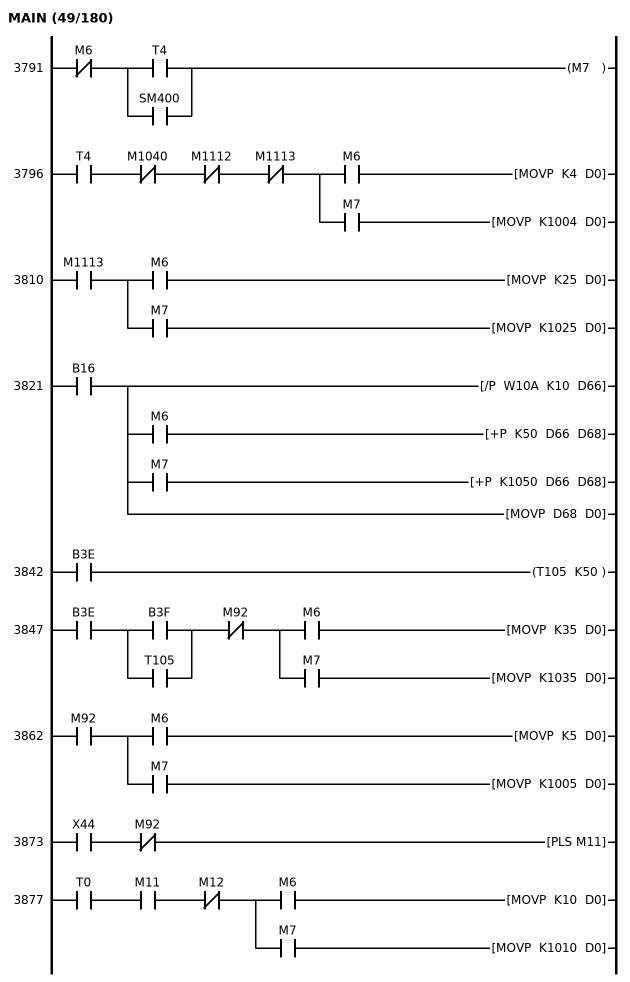
[picture p48: ladder of MAIN, rungs at steps 3791 to 3877]
3791  LDI     M6
      LD      T4
      OR      SM400
      ANB
      OUT     M7
3796  LD      T4
      ANI     M1040
      ANI     M1112
      ANI     M1113
      MPS
      AND     M6
      MOVP    K4 D0
      MPP
      AND     M7
      MOVP    K1004 D0
3810  LD      M1113
      MPS
      AND     M6
      MOVP    K25 D0
      MPP
      AND     M7
      MOVP    K1025 D0
3821  LD      B16
      /P      W10A K10 D66
      MPS
      AND     M6
      +P      K50 D66 D68
      MRD
      AND     M7
      +P      K1050 D66 D68
      MPP
      MOVP    D68 D0
3842  LD      B3E
      OUT     T105 K50
3847  LD      B3E
      LD      B3F
      OR      T105
      ANB
      ANI     M92
      MPS
      AND     M6
      MOVP    K35 D0
      MPP
      AND     M7
      MOVP    K1035 D0
3862  LD      M92
      MPS
      AND     M6
      MOVP    K5 D0
      MPP
      AND     M7
      MOVP    K1005 D0
3873  LD      X44
      ANI     M92
      PLS     M11
3877  LD      T0
      AND     M11
      ANI     M12
      MPS
      AND     M6
      MOVP    K10 D0
      MPP
      AND     M7
      MOVP    K1010 D0
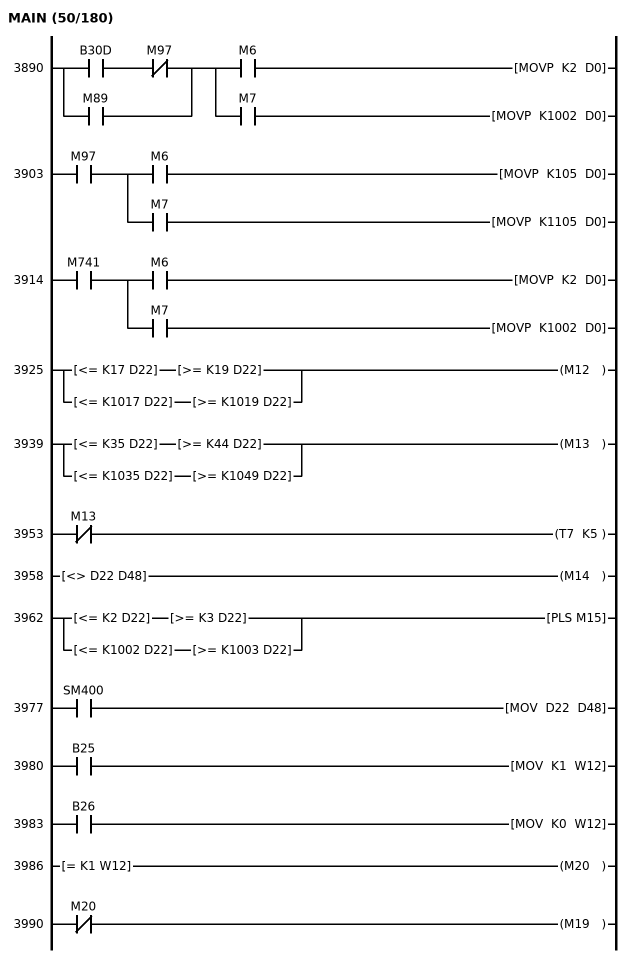
3890  LD      B30D
      ANI     M97
      OR      M89
      MPS
      AND     M6
      MOVP    K2 D0
      MPP
      AND     M7
      MOVP    K1002 D0
3903  LD      M97
      MPS
      AND     M6
      MOVP    K105 D0
      MPP
      AND     M7
      MOVP    K1105 D0
3914  LD      M741
      MPS
      AND     M6
      MOVP    K2 D0
      MPP
      AND     M7
      MOVP    K1002 D0
3925  LD<=    K17 D22
      AND>=   K19 D22
      LD<=    K1017 D22
      AND>=   K1019 D22
      ORB
      OUT     M12
3939  LD<=    K35 D22
      AND>=   K44 D22
      LD<=    K1035 D22
      AND>=   K1049 D22
      ORB
      OUT     M13
3953  LDI     M13
      OUT     T7 K5
3958  LD<>    D22 D48
      OUT     M14
3962  LD<=    K2 D22
      AND>=   K3 D22
      LD<=    K1002 D22
      AND>=   K1003 D22
      ORB
      PLS     M15
3977  LD      SM400
      MOV     D22 D48
3980  LD      B25
      MOV     K1 W12
3983  LD      B26
      MOV     K0 W12
3986  LD=     K1 W12
      OUT     M20
3990  LDI     M20
      OUT     M19
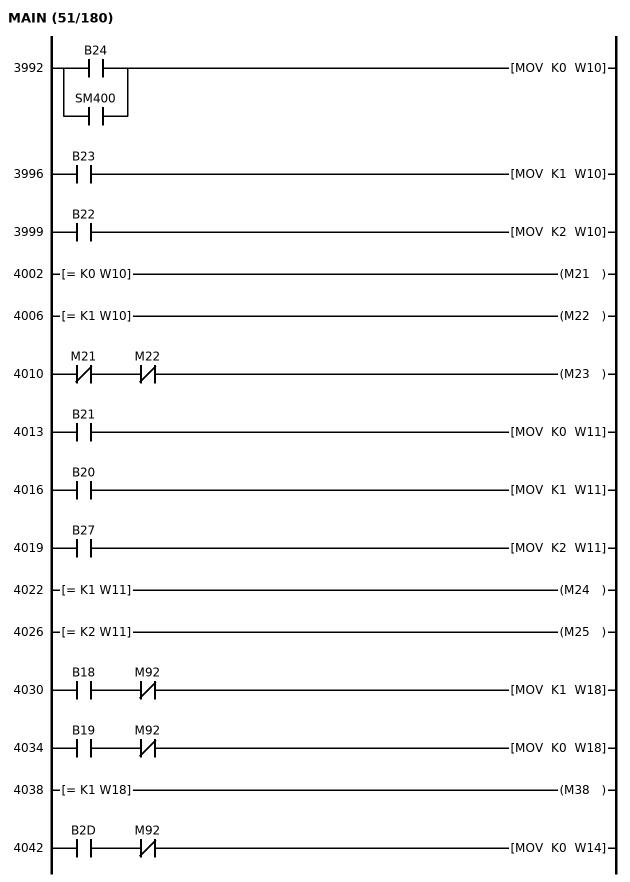
3992  LD      B24
      OR      SM400
      MOV     K0 W10
3996  LD      B23
      MOV     K1 W10
3999  LD      B22
      MOV     K2 W10
4002  LD=     K0 W10
      OUT     M21
4006  LD=     K1 W10
      OUT     M22
4010  LDI     M21
      ANI     M22
      OUT     M23
4013  LD      B21
      MOV     K0 W11
4016  LD      B20
      MOV     K1 W11
4019  LD      B27
      MOV     K2 W11
4022  LD=     K1 W11
      OUT     M24
4026  LD=     K2 W11
      OUT     M25
4030  LD      B18
      ANI     M92
      MOV     K1 W18
4034  LD      B19
      ANI     M92
      MOV     K0 W18
4038  LD=     K1 W18
      OUT     M38
4042  LD      B2D
      ANI     M92
      MOV     K0 W14
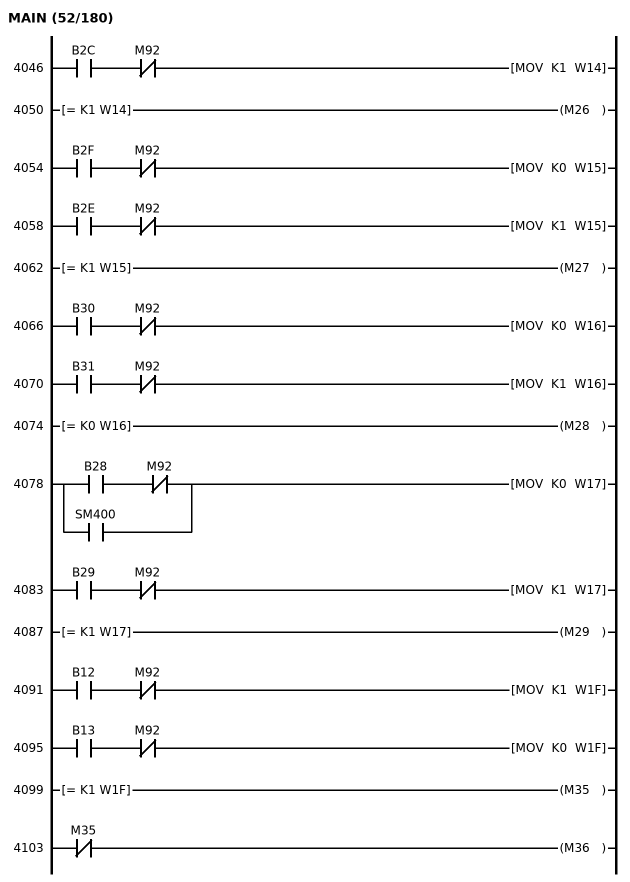
4046  LD      B2C
      ANI     M92
      MOV     K1 W14
4050  LD=     K1 W14
      OUT     M26
4054  LD      B2F
      ANI     M92
      MOV     K0 W15
4058  LD      B2E
      ANI     M92
      MOV     K1 W15
4062  LD=     K1 W15
      OUT     M27
4066  LD      B30
      ANI     M92
      MOV     K0 W16
4070  LD      B31
      ANI     M92
      MOV     K1 W16
4074  LD=     K0 W16
      OUT     M28
4078  LD      B28
      ANI     M92
      OR      SM400
      MOV     K0 W17
4083  LD      B29
      ANI     M92
      MOV     K1 W17
4087  LD=     K1 W17
      OUT     M29
4091  LD      B12
      ANI     M92
      MOV     K1 W1F
4095  LD      B13
      ANI     M92
      MOV     K0 W1F
4099  LD=     K1 W1F
      OUT     M35
4103  LDI     M35
      OUT     M36
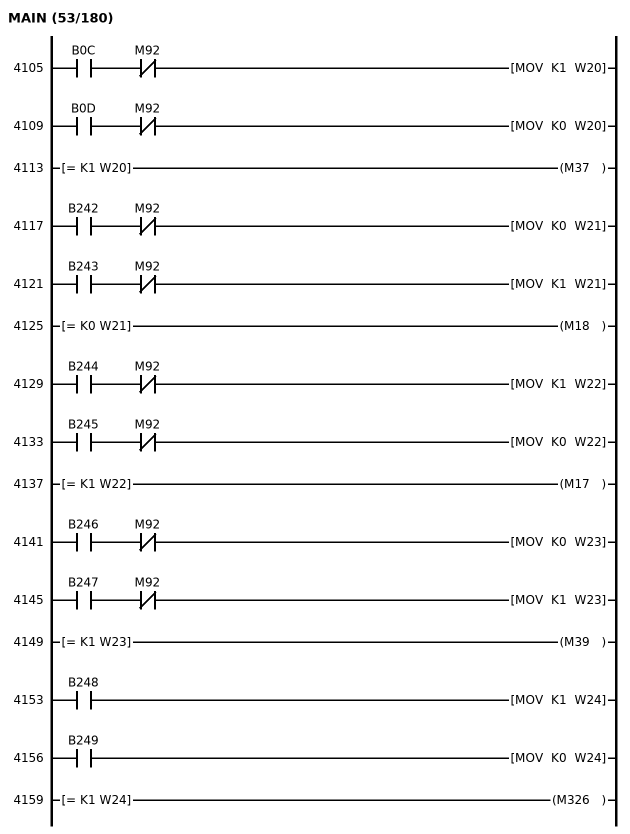
4105  LD      B0C
      ANI     M92
      MOV     K1 W20
4109  LD      B0D
      ANI     M92
      MOV     K0 W20
4113  LD=     K1 W20
      OUT     M37
4117  LD      B242
      ANI     M92
      MOV     K0 W21
4121  LD      B243
      ANI     M92
      MOV     K1 W21
4125  LD=     K0 W21
      OUT     M18
4129  LD      B244
      ANI     M92
      MOV     K1 W22
4133  LD      B245
      ANI     M92
      MOV     K0 W22
4137  LD=     K1 W22
      OUT     M17
4141  LD      B246
      ANI     M92
      MOV     K0 W23
4145  LD      B247
      ANI     M92
      MOV     K1 W23
4149  LD=     K1 W23
      OUT     M39
4153  LD      B248
      MOV     K1 W24
4156  LD      B249
      MOV     K0 W24
4159  LD=     K1 W24
      OUT     M326
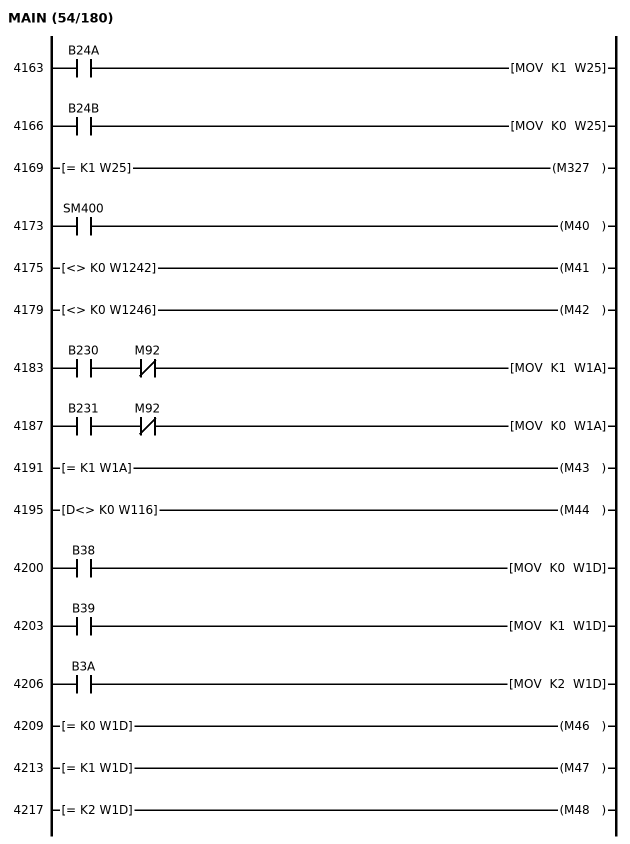
4163  LD      B24A
      MOV     K1 W25
4166  LD      B24B
      MOV     K0 W25
4169  LD=     K1 W25
      OUT     M327
4173  LD      SM400
      OUT     M40
4175  LD<>    K0 W1242
      OUT     M41
4179  LD<>    K0 W1246
      OUT     M42
4183  LD      B230
      ANI     M92
      MOV     K1 W1A
4187  LD      B231
      ANI     M92
      MOV     K0 W1A
4191  LD=     K1 W1A
      OUT     M43
4195  LDD<>   K0 W116
      OUT     M44
4200  LD      B38
      MOV     K0 W1D
4203  LD      B39
      MOV     K1 W1D
4206  LD      B3A
      MOV     K2 W1D
4209  LD=     K0 W1D
      OUT     M46
4213  LD=     K1 W1D
      OUT     M47
4217  LD=     K2 W1D
      OUT     M48
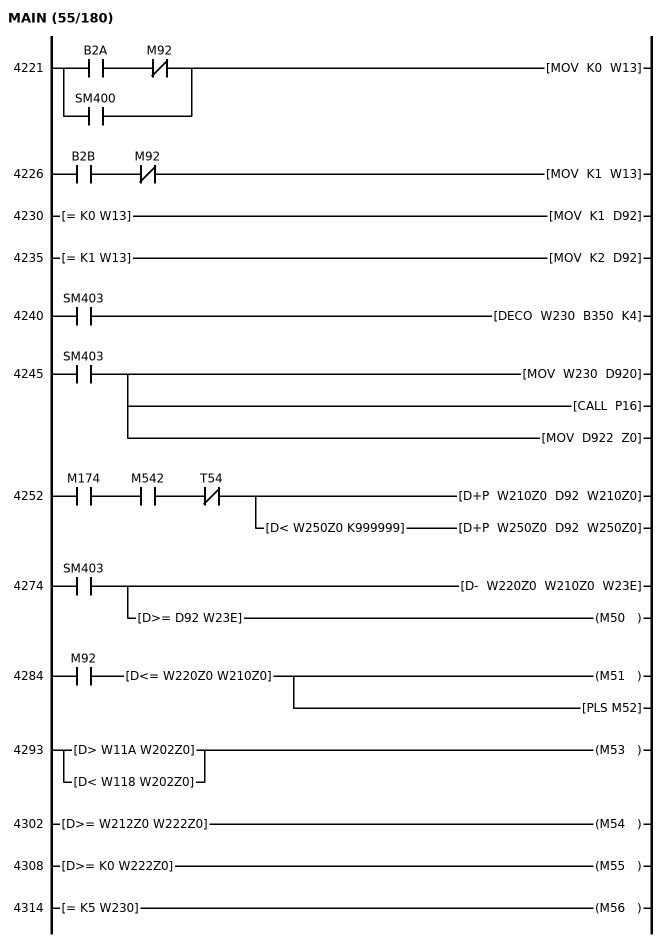
4221  LD      B2A
      ANI     M92
      OR      SM400
      MOV     K0 W13
4226  LD      B2B
      ANI     M92
      MOV     K1 W13
4230  LD=     K0 W13
      MOV     K1 D92
4235  LD=     K1 W13
      MOV     K2 D92
4240  LD      SM403
      DECO    W230 B350 K4
4245  LD      SM403
      MOV     W230 D920
      CALL    P16
      MOV     D922 Z0
4252  LD      M174
      AND     M542
      ANI     T54
      D+P     W210Z0 D92 W210Z0
      ANDD<   W250Z0 K999999
      D+P     W250Z0 D92 W250Z0
4274  LD      SM403
      D-      W220Z0 W210Z0 W23E
      ANDD>=  D92 W23E
      OUT     M50
4284  LD      M92
      ANDD<=  W220Z0 W210Z0
      OUT     M51
      PLS     M52
4293  LDD>    W11A W202Z0
      ORD<    W118 W202Z0
      OUT     M53
4302  LDD>=   W212Z0 W222Z0
      OUT     M54
4308  LDD>=   K0 W222Z0
      OUT     M55
4314  LD=     K5 W230
      OUT     M56
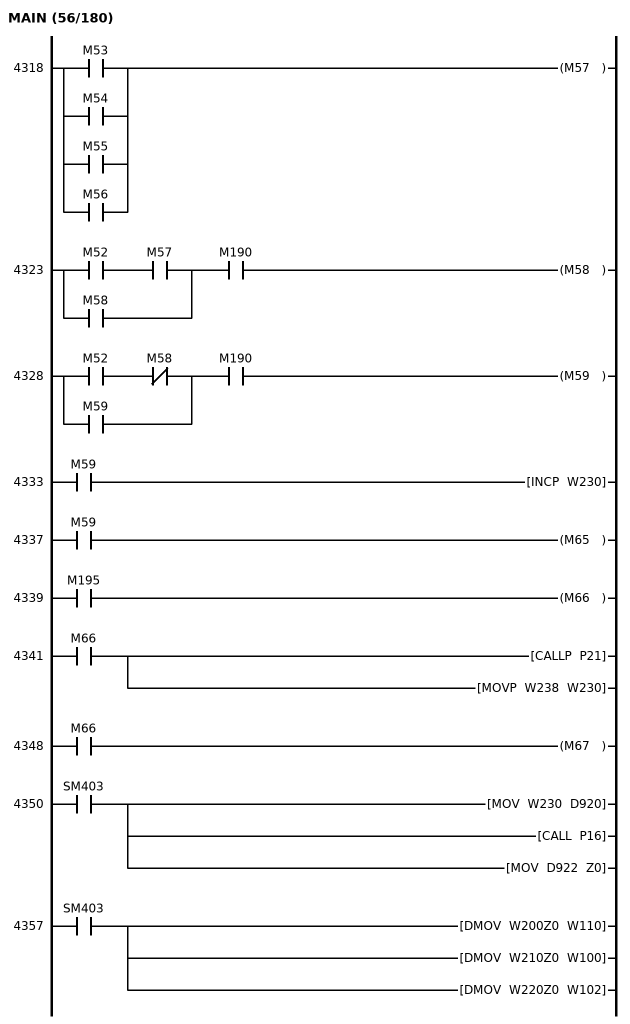
4318  LD      M53
      OR      M54
      OR      M55
      OR      M56
      OUT     M57
4323  LD      M52
      AND     M57
      OR      M58
      AND     M190
      OUT     M58
4328  LD      M52
      ANI     M58
      OR      M59
      AND     M190
      OUT     M59
4333  LD      M59
      INCP    W230
4337  LD      M59
      OUT     M65
4339  LD      M195
      OUT     M66
4341  LD      M66
      CALLP   P21
      MOVP    W238 W230
4348  LD      M66
      OUT     M67
4350  LD      SM403
      MOV     W230 D920
      CALL    P16
      MOV     D922 Z0
4357  LD      SM403
      DMOV    W200Z0 W110
      DMOV    W210Z0 W100
      DMOV    W220Z0 W102
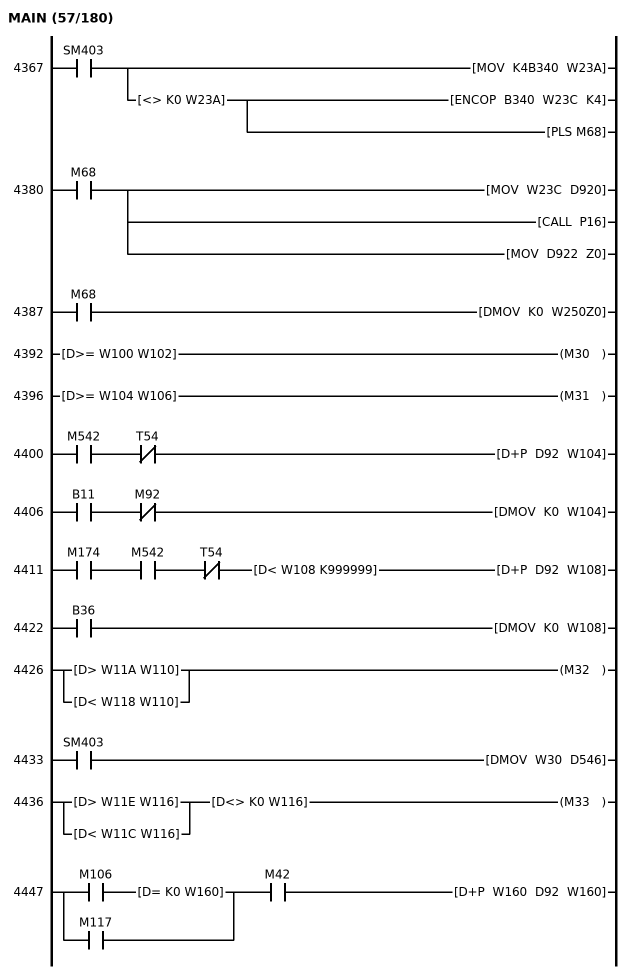
4367  LD      SM403
      MOV     K4B340 W23A
      AND<>   K0 W23A
      ENCOP   B340 W23C K4
      PLS     M68
4380  LD      M68
      MOV     W23C D920
      CALL    P16
      MOV     D922 Z0
4387  LD      M68
      DMOV    K0 W250Z0
4392  LDD>=   W100 W102
      OUT     M30
4396  LDD>=   W104 W106
      OUT     M31
4400  LD      M542
      ANI     T54
      D+P     D92 W104
4406  LD      B11
      ANI     M92
      DMOV    K0 W104
4411  LD      M174
      AND     M542
      ANI     T54
      ANDD<   W108 K999999
      D+P     D92 W108
4422  LD      B36
      DMOV    K0 W108
4426  LDD>    W11A W110
      ORD<    W118 W110
      OUT     M32
4433  LD      SM403
      DMOV    W30 D546
4436  LDD>    W11E W116
      ORD<    W11C W116
      ANDD<>  K0 W116
      OUT     M33
4447  LD      M106
      ANDD=   K0 W160
      OR      M117
      AND     M42
      D+P     W160 D92 W160
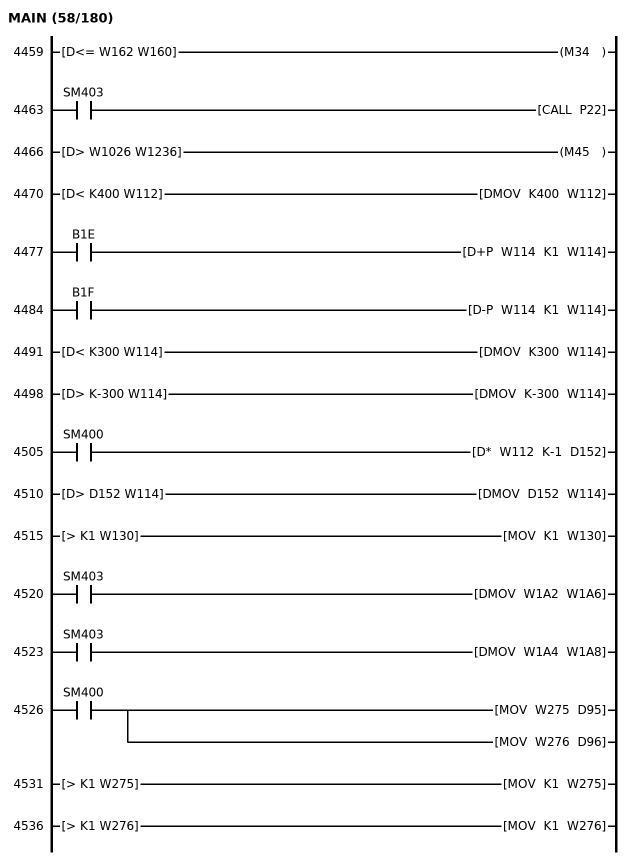
4459  LDD<=   W162 W160
      OUT     M34
4463  LD      SM403
      CALL    P22
4466  LDD>    W1026 W1236
      OUT     M45
4470  LDD<    K400 W112
      DMOV    K400 W112
4477  LD      B1E
      D+P     W114 K1 W114
4484  LD      B1F
      D-P     W114 K1 W114
4491  LDD<    K300 W114
      DMOV    K300 W114
4498  LDD>    K-300 W114
      DMOV    K-300 W114
4505  LD      SM400
      D*      W112 K-1 D152
4510  LDD>    D152 W114
      DMOV    D152 W114
4515  LD>     K1 W130
      MOV     K1 W130
4520  LD      SM403
      DMOV    W1A2 W1A6
4523  LD      SM403
      DMOV    W1A4 W1A8
4526  LD      SM400
      MOV     W275 D95
      MOV     W276 D96
4531  LD>     K1 W275
      MOV     K1 W275
4536  LD>     K1 W276
      MOV     K1 W276
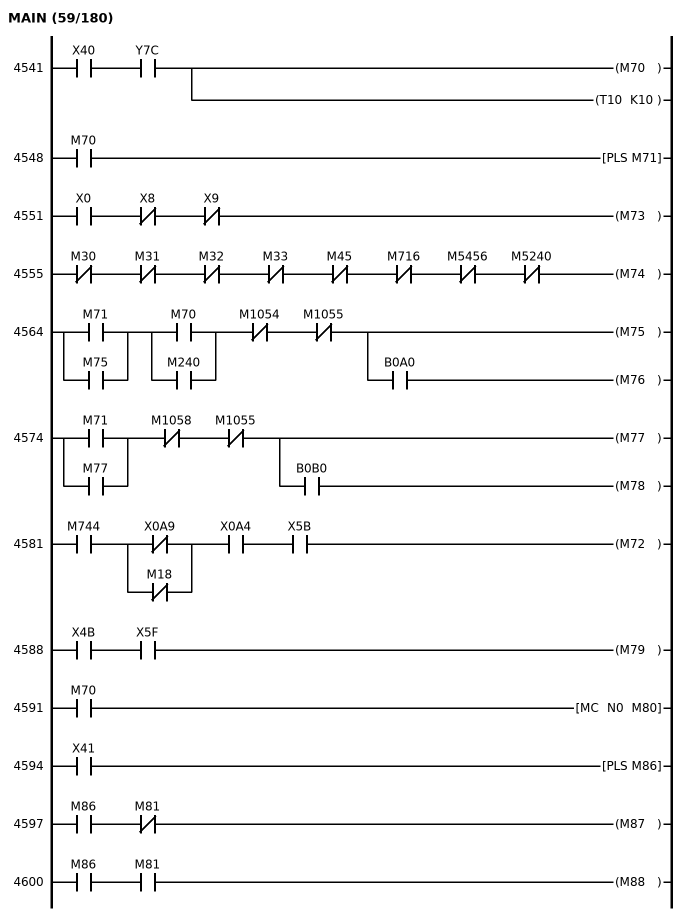
4541  LD      X40
      AND     Y7C
      OUT     M70
      OUT     T10 K10
4548  LD      M70
      PLS     M71
4551  LD      X0
      ANI     X8
      ANI     X9
      OUT     M73
4555  LDI     M30
      ANI     M31
      ANI     M32
      ANI     M33
      ANI     M45
      ANI     M716
      ANI     M5456
      ANI     M5240
      OUT     M74
4564  LD      M71
      OR      M75
      LD      M70
      OR      M240
      ANB
      ANI     M1054
      ANI     M1055
      OUT     M75
      AND     B0A0
      OUT     M76
4574  LD      M71
      OR      M77
      ANI     M1058
      ANI     M1055
      OUT     M77
      AND     B0B0
      OUT     M78
4581  LD      M744
      LDI     X0A9
      ORI     M18
      ANB
      AND     X0A4
      AND     X5B
      OUT     M72
4588  LD      X4B
      AND     X5F
      OUT     M79
4591  LD      M70
      MC      N0 M80
4594  LD      X41
      PLS     M86
4597  LD      M86
      ANI     M81
      OUT     M87
4600  LD      M86
      AND     M81
      OUT     M88
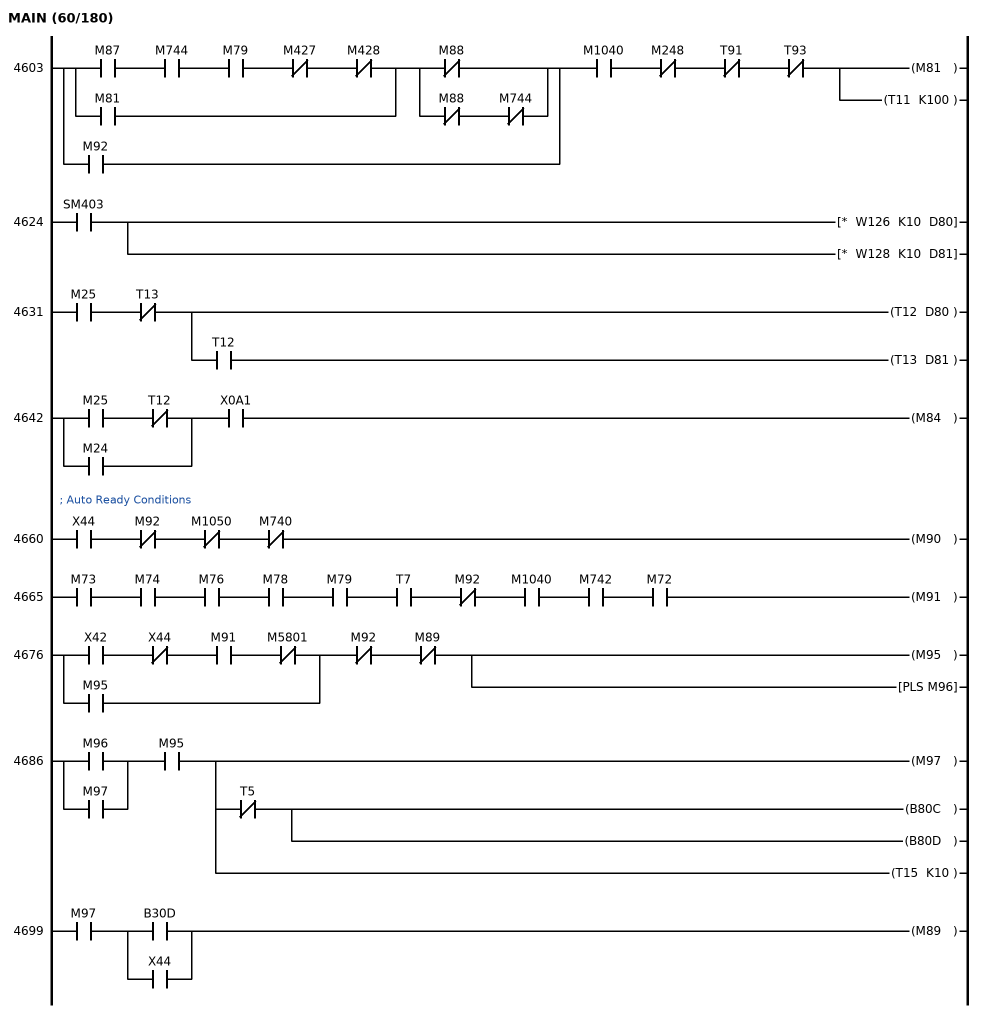
4603  LD      M87
      AND     M744
      AND     M79
      ANI     M427
      ANI     M428
      OR      M81
      LDI     M88
      LDI     M88
      ANI     M744
      ORB
      ANB
      OR      M92
      AND     M1040
      ANI     M248
      ANI     T91
      ANI     T93
      OUT     M81
      OUT     T11 K100
4624  LD      SM403
      *       W126 K10 D80
      *       W128 K10 D81
4631  LD      M25
      ANI     T13
      OUT     T12 D80
      AND     T12
      OUT     T13 D81
4642  LD      M25
      ANI     T12
      OR      M24
      AND     X0A1
      OUT     M84
; Auto Ready Conditions
4660  LD      X44
      ANI     M92
      ANI     M1050
      ANI     M740
      OUT     M90
4665  LD      M73
      AND     M74
      AND     M76
      AND     M78
      AND     M79
      AND     T7
      ANI     M92
      AND     M1040
      AND     M742
      AND     M72
      OUT     M91
4676  LD      X42
      ANI     X44
      AND     M91
      ANI     M5801
      OR      M95
      ANI     M92
      ANI     M89
      OUT     M95
      PLS     M96
4686  LD      M96
      OR      M97
      AND     M95
      OUT     M97
      MPS
      ANI     T5
      OUT     B80C
      OUT     B80D
      MPP
      OUT     T15 K10
4699  LD      M97
      LD      B30D
      OR      X44
      ANB
      OUT     M89
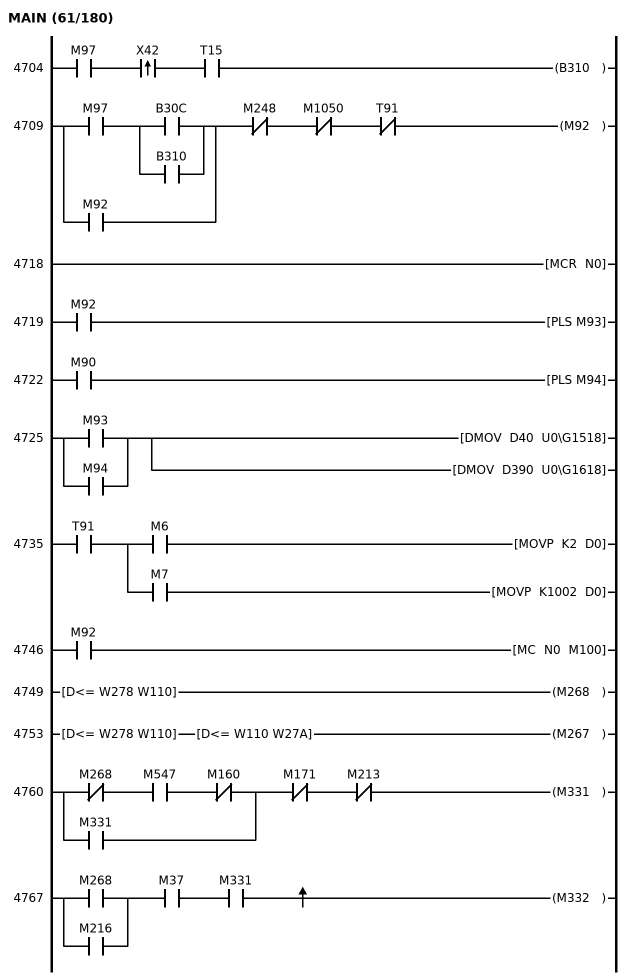
4704  LD      M97
      ANDP    X42
      AND     T15
      OUT     B310
4709  LD      M97
      LD      B30C
      OR      B310
      ANB
      OR      M92
      ANI     M248
      ANI     M1050
      ANI     T91
      OUT     M92
4718  MCR     N0
4719  LD      M92
      PLS     M93
4722  LD      M90
      PLS     M94
4725  LD      M93
      OR      M94
      DMOV    D40 U0\G1518
      DMOV    D390 U0\G1618
4735  LD      T91
      MPS
      AND     M6
      MOVP    K2 D0
      MPP
      AND     M7
      MOVP    K1002 D0
4746  LD      M92
      MC      N0 M100
4749  LDD<=   W278 W110
      OUT     M268
4753  LDD<=   W278 W110
      ANDD<=  W110 W27A
      OUT     M267
4760  LDI     M268
      AND     M547
      ANI     M160
      OR      M331
      ANI     M171
      ANI     M213
      OUT     M331
4767  LD      M268
      OR      M216
      AND     M37
      AND     M331
      MEP
      OUT     M332
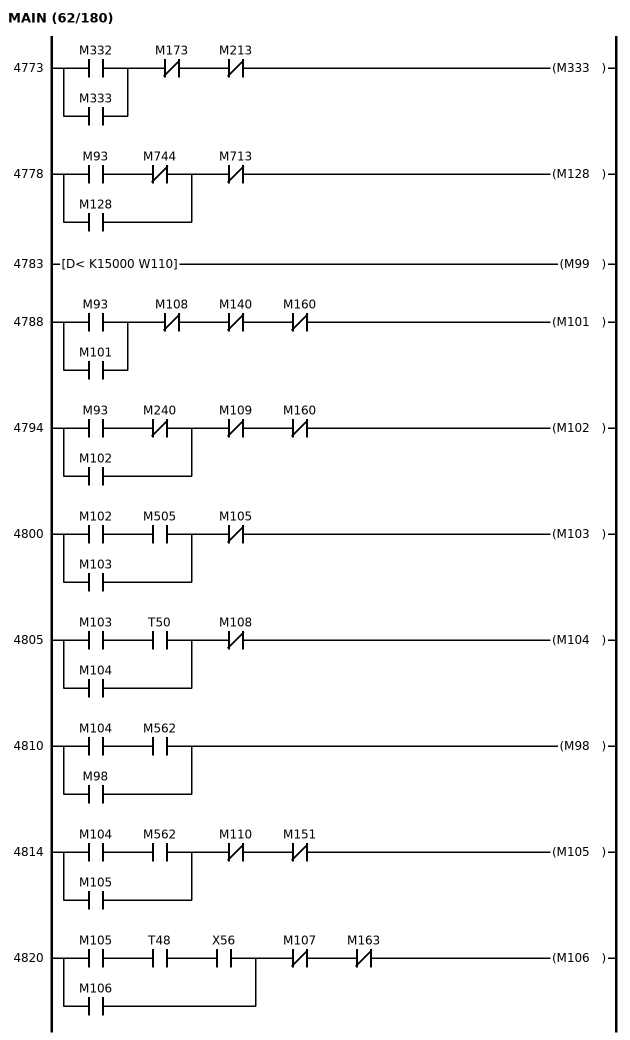
4773  LD      M332
      OR      M333
      ANI     M173
      ANI     M213
      OUT     M333
4778  LD      M93
      ANI     M744
      OR      M128
      ANI     M713
      OUT     M128
4783  LDD<    K15000 W110
      OUT     M99
4788  LD      M93
      OR      M101
      ANI     M108
      ANI     M140
      ANI     M160
      OUT     M101
4794  LD      M93
      ANI     M240
      OR      M102
      ANI     M109
      ANI     M160
      OUT     M102
4800  LD      M102
      AND     M505
      OR      M103
      ANI     M105
      OUT     M103
4805  LD      M103
      AND     T50
      OR      M104
      ANI     M108
      OUT     M104
4810  LD      M104
      AND     M562
      OR      M98
      OUT     M98
4814  LD      M104
      AND     M562
      OR      M105
      ANI     M110
      ANI     M151
      OUT     M105
4820  LD      M105
      AND     T48
      AND     X56
      OR      M106
      ANI     M107
      ANI     M163
      OUT     M106
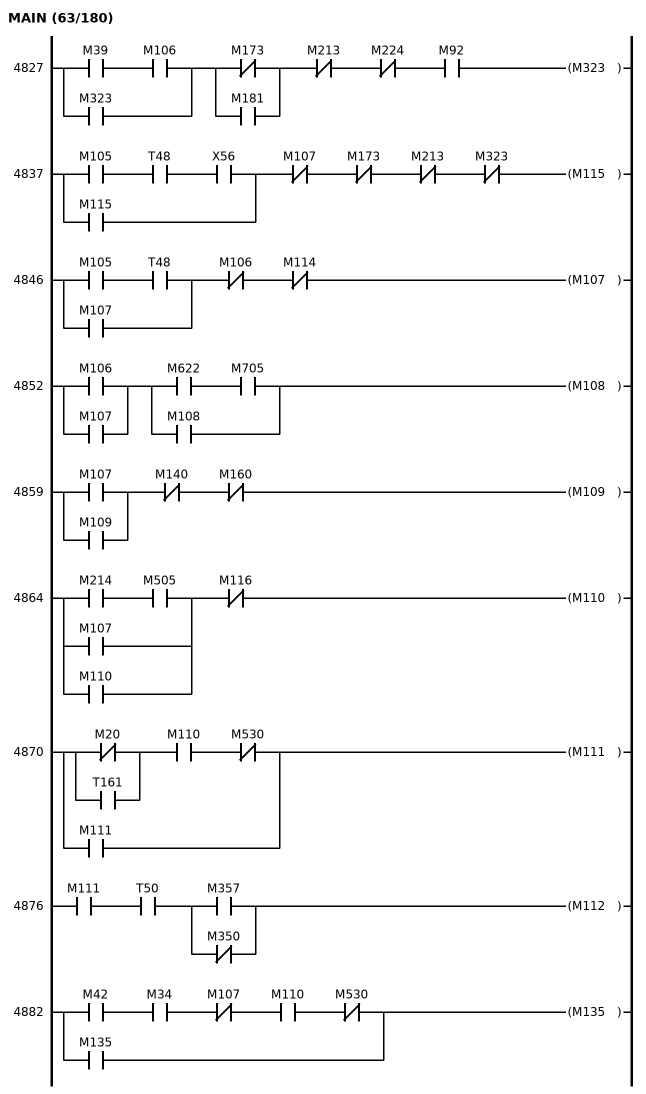
4827  LD      M39
      AND     M106
      OR      M323
      LDI     M173
      OR      M181
      ANB
      ANI     M213
      ANI     M224
      AND     M92
      OUT     M323
4837  LD      M105
      AND     T48
      AND     X56
      OR      M115
      ANI     M107
      ANI     M173
      ANI     M213
      ANI     M323
      OUT     M115
4846  LD      M105
      AND     T48
      OR      M107
      ANI     M106
      ANI     M114
      OUT     M107
4852  LD      M106
      OR      M107
      LD      M622
      AND     M705
      OR      M108
      ANB
      OUT     M108
4859  LD      M107
      OR      M109
      ANI     M140
      ANI     M160
      OUT     M109
4864  LD      M214
      AND     M505
      OR      M107
      OR      M110
      ANI     M116
      OUT     M110
4870  LDI     M20
      OR      T161
      AND     M110
      ANI     M530
      OR      M111
      OUT     M111
4876  LD      M111
      AND     T50
      LD      M357
      ORI     M350
      ANB
      OUT     M112
4882  LD      M42
      AND     M34
      ANI     M107
      AND     M110
      ANI     M530
      OR      M135
      OUT     M135
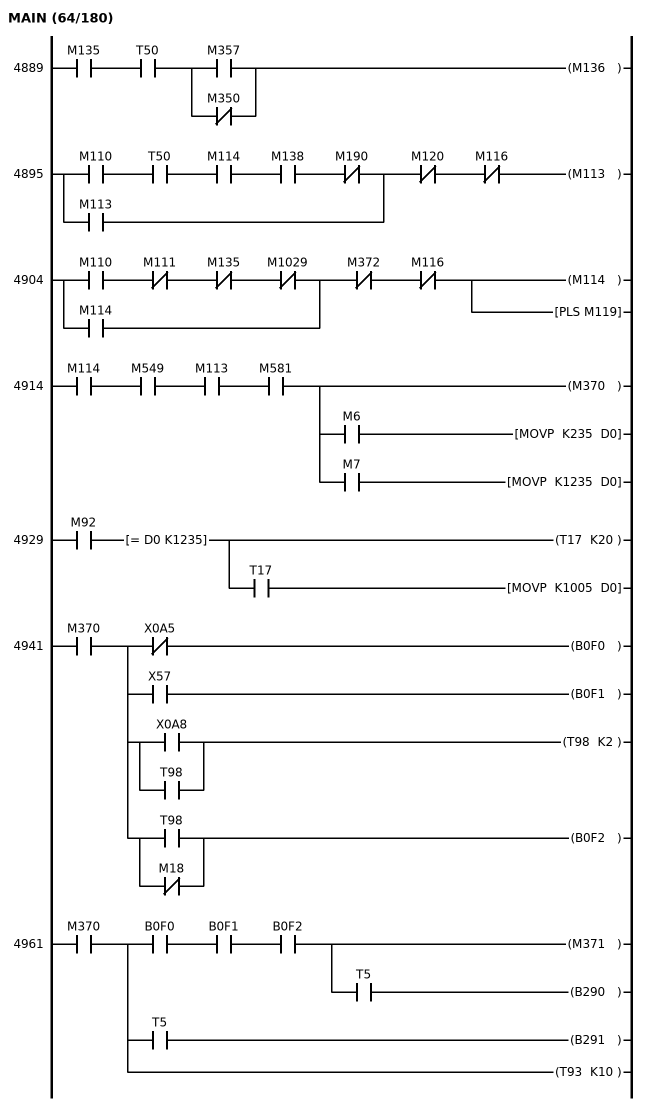
4889  LD      M135
      AND     T50
      LD      M357
      ORI     M350
      ANB
      OUT     M136
4895  LD      M110
      AND     T50
      AND     M114
      AND     M138
      ANI     M190
      OR      M113
      ANI     M120
      ANI     M116
      OUT     M113
4904  LD      M110
      ANI     M111
      ANI     M135
      ANI     M1029
      OR      M114
      ANI     M372
      ANI     M116
      OUT     M114
      PLS     M119
4914  LD      M114
      AND     M549
      AND     M113
      AND     M581
      OUT     M370
      MPS
      AND     M6
      MOVP    K235 D0
      MPP
      AND     M7
      MOVP    K1235 D0
4929  LD      M92
      AND=    D0 K1235
      OUT     T17 K20
      AND     T17
      MOVP    K1005 D0
4941  LD      M370
      MPS
      ANI     X0A5
      OUT     B0F0
      MRD
      AND     X57
      OUT     B0F1
      MRD
      LD      X0A8
      OR      T98
      ANB
      OUT     T98 K2
      MPP
      LD      T98
      ORI     M18
      ANB
      OUT     B0F2
4961  LD      M370
      MPS
      AND     B0F0
      AND     B0F1
      AND     B0F2
      OUT     M371
      AND     T5
      OUT     B290
      MRD
      AND     T5
      OUT     B291
      MPP
      OUT     T93 K10
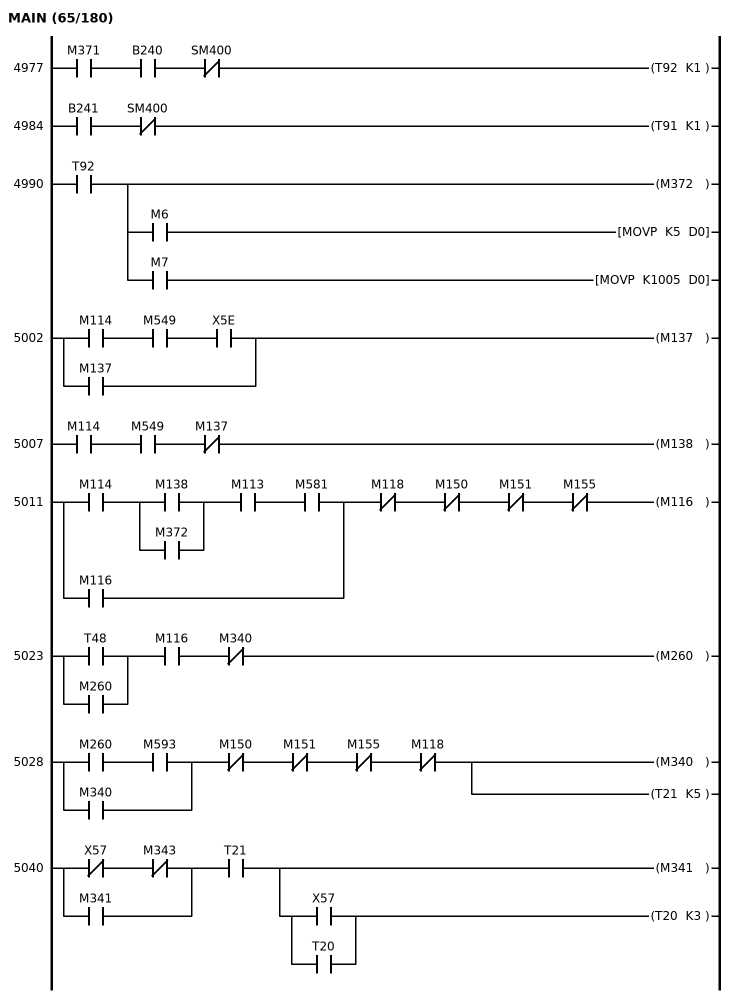
4977  LD      M371
      AND     B240
      ANI     SM400
      OUT     T92 K1
4984  LD      B241
      ANI     SM400
      OUT     T91 K1
4990  LD      T92
      OUT     M372
      MPS
      AND     M6
      MOVP    K5 D0
      MPP
      AND     M7
      MOVP    K1005 D0
5002  LD      M114
      AND     M549
      AND     X5E
      OR      M137
      OUT     M137
5007  LD      M114
      AND     M549
      ANI     M137
      OUT     M138
5011  LD      M114
      LD      M138
      OR      M372
      ANB
      AND     M113
      AND     M581
      OR      M116
      ANI     M118
      ANI     M150
      ANI     M151
      ANI     M155
      OUT     M116
5023  LD      T48
      OR      M260
      AND     M116
      ANI     M340
      OUT     M260
5028  LD      M260
      AND     M593
      OR      M340
      ANI     M150
      ANI     M151
      ANI     M155
      ANI     M118
      OUT     M340
      OUT     T21 K5
5040  LDI     X57
      ANI     M343
      OR      M341
      AND     T21
      OUT     M341
      LD      X57
      OR      T20
      ANB
      OUT     T20 K3
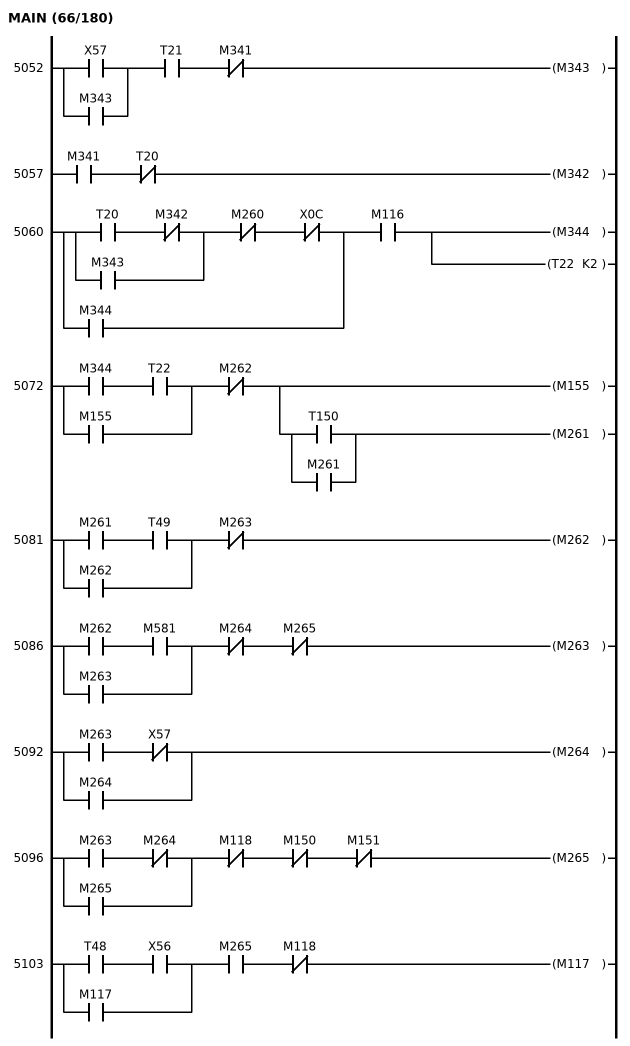
5052  LD      X57
      OR      M343
      AND     T21
      ANI     M341
      OUT     M343
5057  LD      M341
      ANI     T20
      OUT     M342
5060  LD      T20
      ANI     M342
      OR      M343
      ANI     M260
      ANI     X0C
      OR      M344
      AND     M116
      OUT     M344
      OUT     T22 K2
5072  LD      M344
      AND     T22
      OR      M155
      ANI     M262
      OUT     M155
      LD      T150
      OR      M261
      ANB
      OUT     M261
5081  LD      M261
      AND     T49
      OR      M262
      ANI     M263
      OUT     M262
5086  LD      M262
      AND     M581
      OR      M263
      ANI     M264
      ANI     M265
      OUT     M263
5092  LD      M263
      ANI     X57
      OR      M264
      OUT     M264
5096  LD      M263
      ANI     M264
      OR      M265
      ANI     M118
      ANI     M150
      ANI     M151
      OUT     M265
5103  LD      T48
      AND     X56
      OR      M117
      AND     M265
      ANI     M118
      OUT     M117
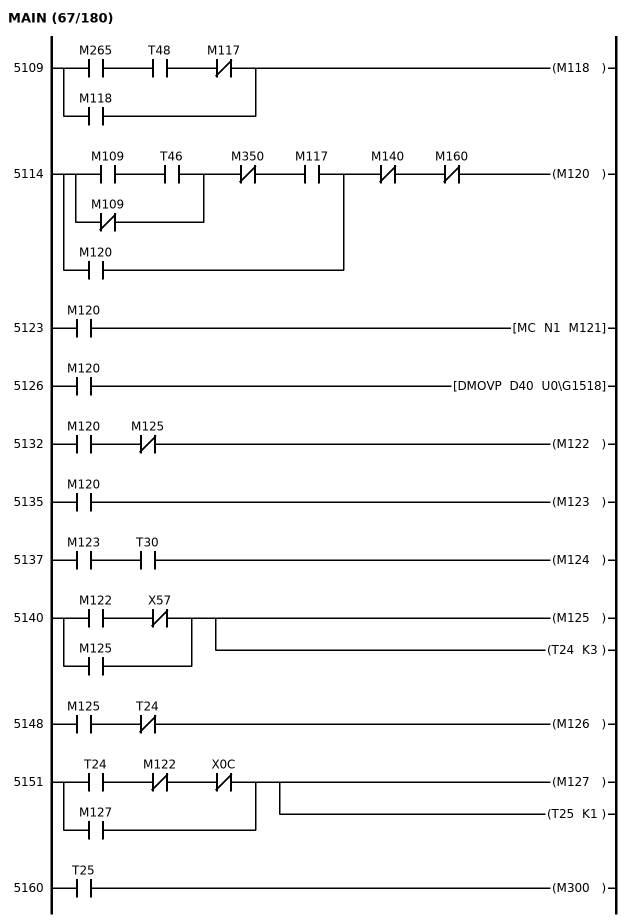
5109  LD      M265
      AND     T48
      ANI     M117
      OR      M118
      OUT     M118
5114  LD      M109
      AND     T46
      ORI     M109
      ANI     M350
      AND     M117
      OR      M120
      ANI     M140
      ANI     M160
      OUT     M120
5123  LD      M120
      MC      N1 M121
5126  LD      M120
      DMOVP   D40 U0\G1518
5132  LD      M120
      ANI     M125
      OUT     M122
5135  LD      M120
      OUT     M123
5137  LD      M123
      AND     T30
      OUT     M124
5140  LD      M122
      ANI     X57
      OR      M125
      OUT     M125
      OUT     T24 K3
5148  LD      M125
      ANI     T24
      OUT     M126
5151  LD      T24
      ANI     M122
      ANI     X0C
      OR      M127
      OUT     M127
      OUT     T25 K1
5160  LD      T25
      OUT     M300
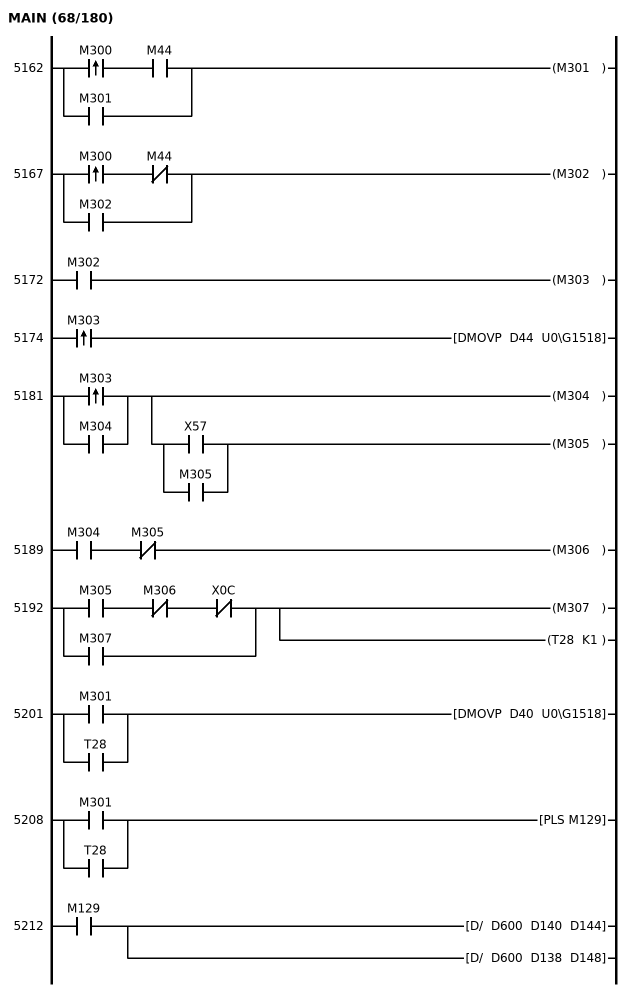
5162  LDP     M300
      AND     M44
      OR      M301
      OUT     M301
5167  LDP     M300
      ANI     M44
      OR      M302
      OUT     M302
5172  LD      M302
      OUT     M303
5174  LDP     M303
      DMOVP   D44 U0\G1518
5181  LDP     M303
      OR      M304
      OUT     M304
      LD      X57
      OR      M305
      ANB
      OUT     M305
5189  LD      M304
      ANI     M305
      OUT     M306
5192  LD      M305
      ANI     M306
      ANI     X0C
      OR      M307
      OUT     M307
      OUT     T28 K1
5201  LD      M301
      OR      T28
      DMOVP   D40 U0\G1518
5208  LD      M301
      OR      T28
      PLS     M129
5212  LD      M129
      D/      D600 D140 D144
      D/      D600 D138 D148
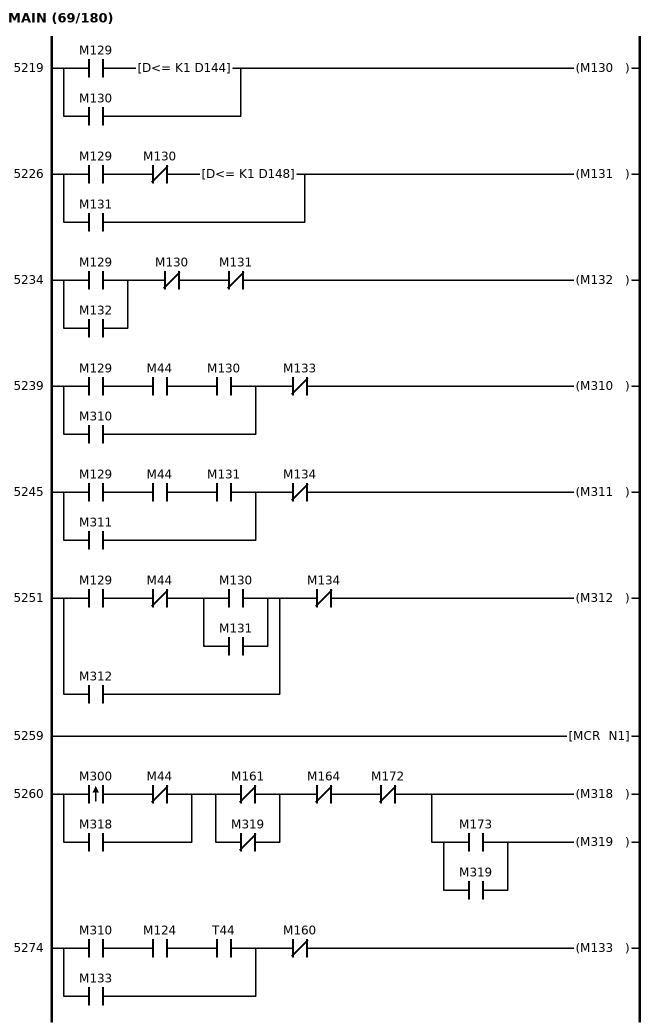
5219  LD      M129
      ANDD<=  K1 D144
      OR      M130
      OUT     M130
5226  LD      M129
      ANI     M130
      ANDD<=  K1 D148
      OR      M131
      OUT     M131
5234  LD      M129
      OR      M132
      ANI     M130
      ANI     M131
      OUT     M132
5239  LD      M129
      AND     M44
      AND     M130
      OR      M310
      ANI     M133
      OUT     M310
5245  LD      M129
      AND     M44
      AND     M131
      OR      M311
      ANI     M134
      OUT     M311
5251  LD      M129
      ANI     M44
      LD      M130
      OR      M131
      ANB
      OR      M312
      ANI     M134
      OUT     M312
5259  MCR     N1
5260  LDP     M300
      ANI     M44
      OR      M318
      LDI     M161
      ORI     M319
      ANB
      ANI     M164
      ANI     M172
      OUT     M318
      LD      M173
      OR      M319
      ANB
      OUT     M319
5274  LD      M310
      AND     M124
      AND     T44
      OR      M133
      ANI     M160
      OUT     M133
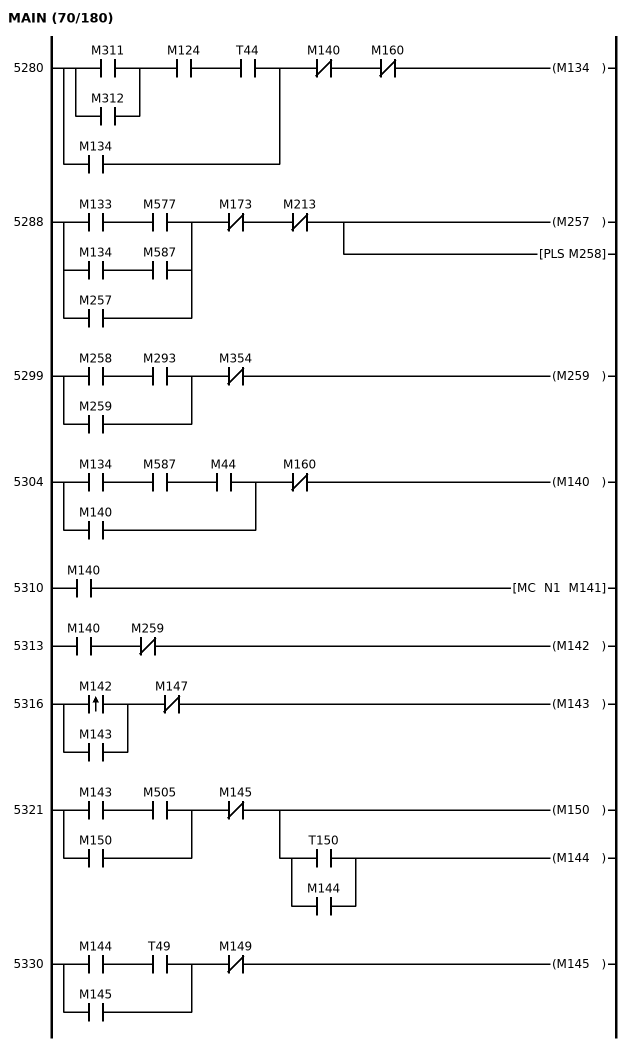
5280  LD      M311
      OR      M312
      AND     M124
      AND     T44
      OR      M134
      ANI     M140
      ANI     M160
      OUT     M134
5288  LD      M133
      AND     M577
      LD      M134
      AND     M587
      ORB
      OR      M257
      ANI     M173
      ANI     M213
      OUT     M257
      PLS     M258
5299  LD      M258
      AND     M293
      OR      M259
      ANI     M354
      OUT     M259
5304  LD      M134
      AND     M587
      AND     M44
      OR      M140
      ANI     M160
      OUT     M140
5310  LD      M140
      MC      N1 M141
5313  LD      M140
      ANI     M259
      OUT     M142
5316  LDP     M142
      OR      M143
      ANI     M147
      OUT     M143
5321  LD      M143
      AND     M505
      OR      M150
      ANI     M145
      OUT     M150
      LD      T150
      OR      M144
      ANB
      OUT     M144
5330  LD      M144
      AND     T49
      OR      M145
      ANI     M149
      OUT     M145
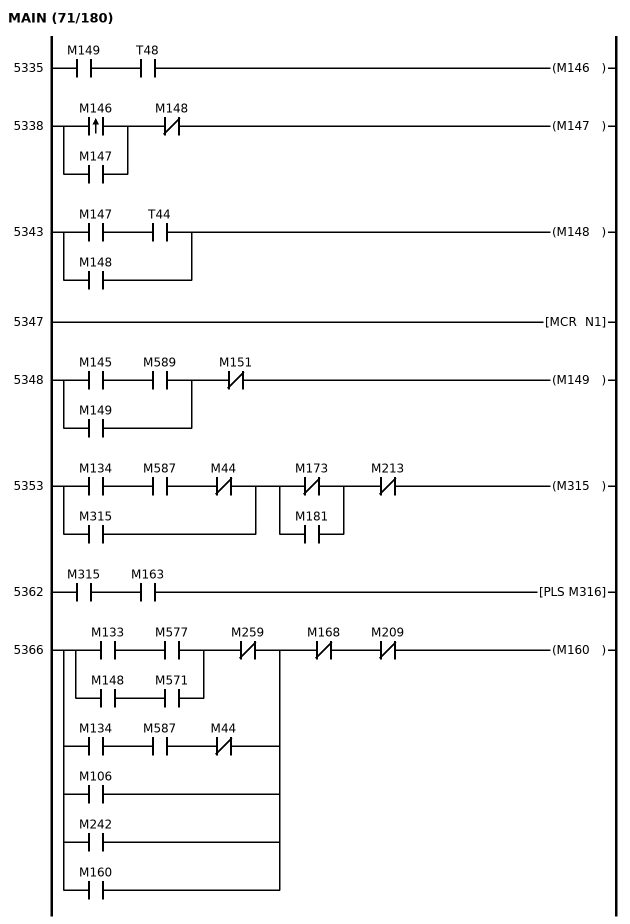
5335  LD      M149
      AND     T48
      OUT     M146
5338  LDP     M146
      OR      M147
      ANI     M148
      OUT     M147
5343  LD      M147
      AND     T44
      OR      M148
      OUT     M148
5347  MCR     N1
5348  LD      M145
      AND     M589
      OR      M149
      ANI     M151
      OUT     M149
5353  LD      M134
      AND     M587
      ANI     M44
      OR      M315
      LDI     M173
      OR      M181
      ANB
      ANI     M213
      OUT     M315
5362  LD      M315
      AND     M163
      PLS     M316
5366  LD      M133
      AND     M577
      LD      M148
      AND     M571
      ORB
      ANI     M259
      LD      M134
      AND     M587
      ANI     M44
      ORB
      OR      M106
      OR      M242
      OR      M160
      ANI     M168
      ANI     M209
      OUT     M160
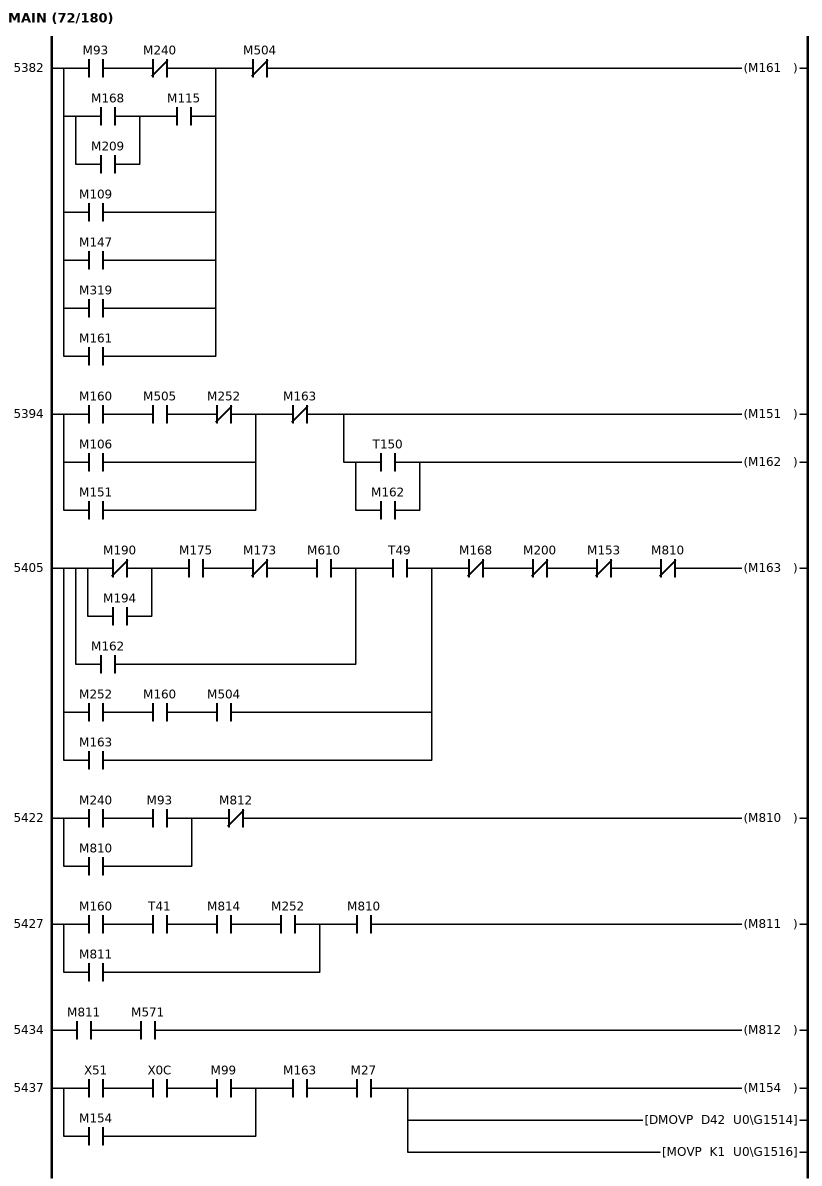
5382  LD      M93
      ANI     M240
      LD      M168
      OR      M209
      AND     M115
      ORB
      OR      M109
      OR      M147
      OR      M319
      OR      M161
      ANI     M504
      OUT     M161
5394  LD      M160
      AND     M505
      ANI     M252
      OR      M106
      OR      M151
      ANI     M163
      OUT     M151
      LD      T150
      OR      M162
      ANB
      OUT     M162
5405  LDI     M190
      OR      M194
      AND     M175
      ANI     M173
      AND     M610
      OR      M162
      AND     T49
      LD      M252
      AND     M160
      AND     M504
      ORB
      OR      M163
      ANI     M168
      ANI     M200
      ANI     M153
      ANI     M810
      OUT     M163
5422  LD      M240
      AND     M93
      OR      M810
      ANI     M812
      OUT     M810
5427  LD      M160
      AND     T41
      AND     M814
      AND     M252
      OR      M811
      AND     M810
      OUT     M811
5434  LD      M811
      AND     M571
      OUT     M812
5437  LD      X51
      AND     X0C
      AND     M99
      OR      M154
      AND     M163
      AND     M27
      OUT     M154
      DMOVP   D42 U0\G1514
      MOVP    K1 U0\G1516
